// TIA Portal project "WindTurbineOperativeState" (V17)
// Operation state control system of wind turbine

(* hardware
DEVICE "S7-1200 station_1"  S7-1200 Station
   slot 0: "Rack_0"  S7-1200 Rack  Rack  V1.0
   slot 1: "PLC_1"  CPU 1211C DC/DC/DC  6ES7 211-1AE40-0XB0  V4.5
*)

// ===== PLC "PLC_1"  CPU 1211C DC/DC/DC =====

VAR_GLOBAL   // PLC tag table "Default tag table"
   "_WindSpeed_AI" AT %IW64 : Int;
   "_TurbineRotation_AI" AT %IW66 : Int;
   "EmergencyStop_BTN" AT %I0.0 : Bool;
   "BlockState_BTN" AT %I0.1 : Bool;
   "ParkingBrake" AT %Q0.0 : Bool;
   "PitchBrake" AT %Q0.1 : Bool;
   "GeneratorTrip" AT %Q0.2 : Bool;
   "_BlockState" AT %M0.0 : Bool;
   "WebError" AT %MW0 : Int;
END_VAR

VAR_GLOBAL CONSTANT   // PLC tag table "Default tag table"
   "_ParkBrake" : Byte := 0;
   "_Startup" : Byte := 1;
   "_Generating" : Byte := 2;
   "_PitchBrake" : Byte := 3;
END_VAR

DATA_BLOCK "CompOnDuration_DB_13"   // DB1
{ S7_Optimized_Access := 'TRUE' }
VERSION : 0.1
// stored: InstanceOfName CompOnDuration
"CompOnDuration"
BEGIN
END_DATA_BLOCK

DATA_BLOCK "CompOnDuration_DB_01"   // DB2
{ S7_Optimized_Access := 'TRUE' }
VERSION : 0.1
// stored: InstanceOfName CompOnDuration
"CompOnDuration"
BEGIN
END_DATA_BLOCK

DATA_BLOCK "CompOnDuration_DB_02"   // DB3
{ S7_Optimized_Access := 'TRUE' }
VERSION : 0.1
// stored: InstanceOfName CompOnDuration
"CompOnDuration"
BEGIN
END_DATA_BLOCK

DATA_BLOCK "CompOnDuration_DB_03"   // DB4
{ S7_Optimized_Access := 'TRUE' }
VERSION : 0.1
// stored: InstanceOfName CompOnDuration
"CompOnDuration"
BEGIN
END_DATA_BLOCK

DATA_BLOCK "CompOnDuration_DB_04"   // DB5
{ S7_Optimized_Access := 'TRUE' }
VERSION : 0.1
// stored: InstanceOfName CompOnDuration
"CompOnDuration"
BEGIN
END_DATA_BLOCK

DATA_BLOCK "CompOnDuration_DB_05"   // DB6
{ S7_Optimized_Access := 'TRUE' }
VERSION : 0.1
// stored: InstanceOfName CompOnDuration
"CompOnDuration"
BEGIN
END_DATA_BLOCK

DATA_BLOCK "CompOnDuration_DB_06"   // DB7
{ S7_Optimized_Access := 'TRUE' }
VERSION : 0.1
// stored: InstanceOfName CompOnDuration
"CompOnDuration"
BEGIN
END_DATA_BLOCK

DATA_BLOCK "CompOnDuration_DB_07"   // DB8
{ S7_Optimized_Access := 'TRUE' }
VERSION : 0.1
// stored: InstanceOfName CompOnDuration
"CompOnDuration"
BEGIN
END_DATA_BLOCK

DATA_BLOCK "CompOnDuration_DB_08"   // DB9
{ S7_Optimized_Access := 'TRUE' }
VERSION : 0.1
// stored: InstanceOfName CompOnDuration
"CompOnDuration"
BEGIN
END_DATA_BLOCK

DATA_BLOCK "CompOnDuration_DB_09"   // DB10
{ S7_Optimized_Access := 'TRUE' }
VERSION : 0.1
// stored: InstanceOfName CompOnDuration
"CompOnDuration"
BEGIN
END_DATA_BLOCK

DATA_BLOCK "CompOnDuration_DB_10"   // DB11
{ S7_Optimized_Access := 'TRUE' }
VERSION : 0.1
// stored: InstanceOfName CompOnDuration
"CompOnDuration"
BEGIN
END_DATA_BLOCK

DATA_BLOCK "CompOnDuration_DB_11"   // DB12
{ S7_Optimized_Access := 'TRUE' }
VERSION : 0.1
// stored: InstanceOfName CompOnDuration
"CompOnDuration"
BEGIN
END_DATA_BLOCK

DATA_BLOCK "CompOnDuration_DB_12"   // DB13
{ S7_Optimized_Access := 'TRUE' }
VERSION : 0.1
// stored: InstanceOfName CompOnDuration
"CompOnDuration"
BEGIN
END_DATA_BLOCK

DATA_BLOCK "ModBus_DB"   // DB14
{ S7_Optimized_Access := 'TRUE' }
VERSION : 0.1
   VAR
      CONNECT : TCON_IP_v4;
      ERROR : Bool;
      STATUS : Word;
   END_VAR
BEGIN
   CONNECT.InterfaceId := 64;
   CONNECT.LocalPort := 502;
   CONNECT.ID := 1;
   CONNECT.ConnectionType := 11;
END_DATA_BLOCK

DATA_BLOCK "Hold_Reg"   // DB16
{ S7_Optimized_Access := 'FALSE' }
VERSION : 0.1
   VAR
      TurbineState : Byte;
      BlockState_MB : Bool := false;
      vWind : Real;
      wTurbine : Real;
      vWind_CutInLow : Real := 4.0;
      vWind_CutInUp : Real := 18.0;
      vWind_CutOut : Real := 20.0;
      wTurbine_CutIn : Real := 11.0;
      wTurbine_CutOut : Real := 22.0;
      wTurbine_Parking : Real := 2.0;
      vWind_zero : Int := 34;   // Ofset for 0 reference dac0
      vWind_max : Int := 25051;   // Ofset for 1023 reference dac0
      vWind_gain : Real := 102.3;   // Scale to SI value for "vWind_AI"
      wTurbine_zero : Int := 0;   // Ofset for 0 reference dac1
      wTurbine_max : Int := 25151;   // Ofset for 1023 reference dac1
      wTurbine_gain : Real := 31.0;   // Scale to SI value for "wTurbine_AI"
      time_0 : Time := T#700ms;
      time_1 : Time := T#1.5s;
      time_2 : Time := T#3s;
   END_VAR
BEGIN
END_DATA_BLOCK

FUNCTION_BLOCK "CompOnDuration"   // FB1, LAD
{ S7_Optimized_Access := 'TRUE' }
VERSION : 0.1
// Compare if #A > #B for a duration of at least #Time set #Q
   VAR_INPUT
      "A" : Real;
      "B" : Real;
      "Time" : Time;
   END_VAR
   VAR_OUTPUT
      Q : Bool;
   END_VAR
   VAR
      "IEC_Timer_Multi-Instance" : TON_TIME;
   END_VAR
BEGIN

REGION Network 1
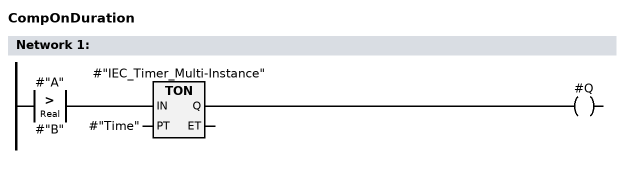
   #"IEC_Timer_Multi-Instance"(IN := #"A" > #"B", PT := #"Time");   // TON
   #Q := #"IEC_Timer_Multi-Instance".Q;
END_REGION
END_FUNCTION_BLOCK

ORGANIZATION_BLOCK "Main"   // OB1, LAD, ProgramCycle
TITLE = "Main Program Sweep (Cycle)"
{ S7_Optimized_Access := 'TRUE' }
VERSION : 0.1
// State machine turbine operation
   VAR_INPUT
      Initial_Call : Bool;   // Initial call of this OB
      Remanence : Bool;   // =True, if remanent data are available
   END_VAR
   VAR_TEMP
      "0to1_1" : Bool;
      "0to1_2" : Bool;
      "1to2" : Bool;
      "1to3_1" : Bool;
      "1to3_2" : Bool;
      "2to3_1" : Bool;
      "2to3_2" : Bool;
      "2to3_3" : Bool;
      "2to3_4" : Bool;
      "3to1_1" : Bool;
      "3to1_2" : Bool;
      "3to1_3" : Bool;
      "3to0" : Bool;
      Norm_vWind : Real;
      Norm_wTurbine : Real;
   END_VAR
   VAR_TEMP   // added for the SCL form of the ladder/FBD networks
      _w1 : Bool;
      _w2 : Bool;
      _w3 : Bool;
      _w4 : Bool;
   END_VAR
BEGIN

REGION Network 1: vWind conversion
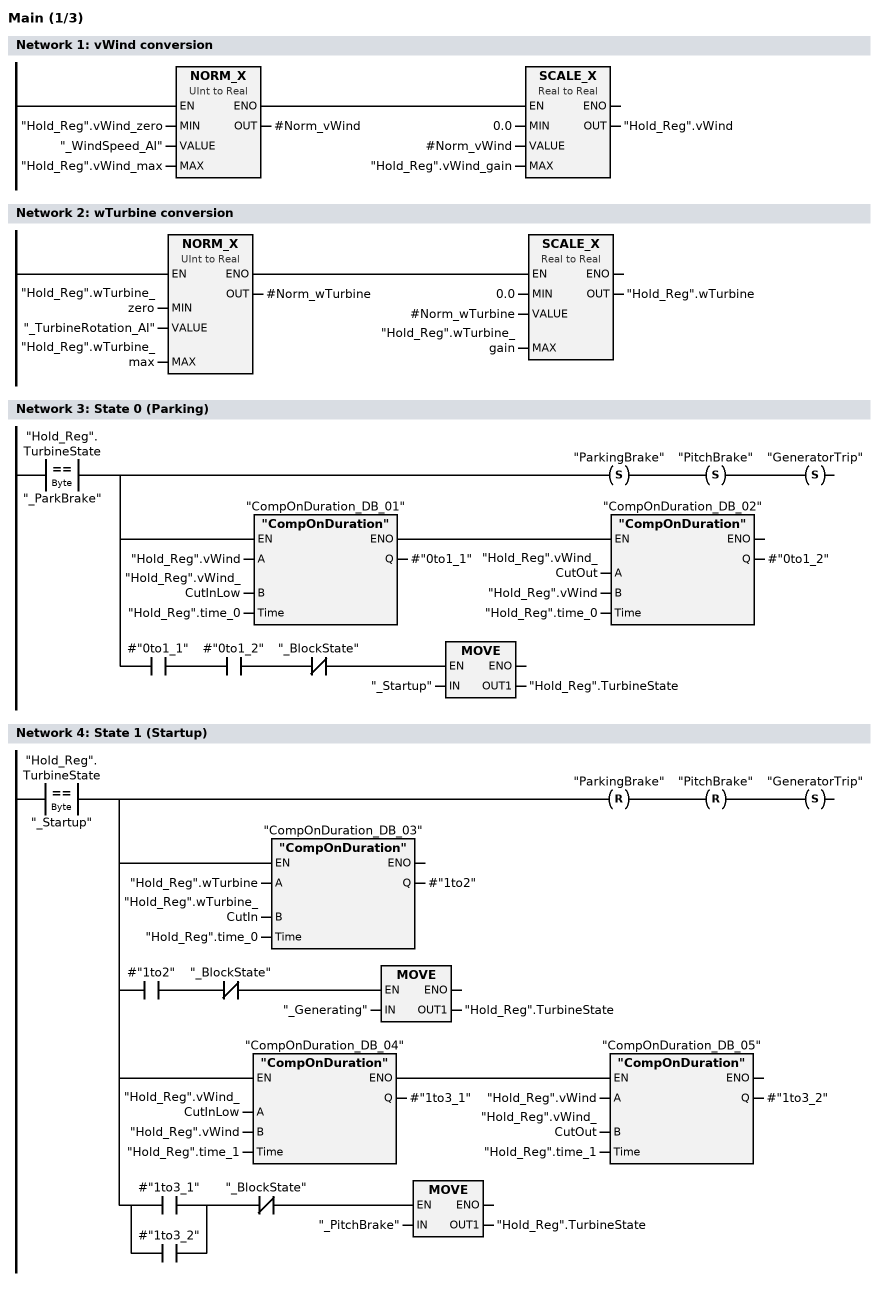
   RUNG wire#powerrail
      { S7_Templates := "[SrcType := UInt, DestType := Real]" } Normalize(min := "Hold_Reg".vWind_zero, value := "_WindSpeed_AI", max := "Hold_Reg".vWind_max, out => #Norm_vWind)
      { S7_Templates := "[SrcType := Real, DestType := Real]" } Scale(min := 0.0, value := #Norm_vWind, max := "Hold_Reg".vWind_gain, out => "Hold_Reg".vWind)
   END_RUNG
   // the same network as SCL:
   #Norm_vWind := NORM_X(MIN := "Hold_Reg".vWind_zero, VALUE := "_WindSpeed_AI", MAX := "Hold_Reg".vWind_max);
   "Hold_Reg".vWind := SCALE_X(MIN := 0.0, VALUE := #Norm_vWind, MAX := "Hold_Reg".vWind_gain);
END_REGION

REGION Network 2: wTurbine conversion
   RUNG wire#powerrail
      { S7_Templates := "[SrcType := UInt, DestType := Real]" } Normalize(min := "Hold_Reg".wTurbine_zero, value := "_TurbineRotation_AI", max := "Hold_Reg".wTurbine_max, out => #Norm_wTurbine)
      { S7_Templates := "[SrcType := Real, DestType := Real]" } Scale(min := 0.0, value := #Norm_wTurbine, max := "Hold_Reg".wTurbine_gain, out => "Hold_Reg".wTurbine)
   END_RUNG
   // the same network as SCL:
   #Norm_wTurbine := NORM_X(MIN := "Hold_Reg".wTurbine_zero, VALUE := "_TurbineRotation_AI", MAX := "Hold_Reg".wTurbine_max);
   "Hold_Reg".wTurbine := SCALE_X(MIN := 0.0, VALUE := #Norm_wTurbine, MAX := "Hold_Reg".wTurbine_gain);
END_REGION

REGION Network 3: State 0 (Parking)
   RUNG wire#powerrail
      { S7_Templates := "SrcType := Byte" } EQ_Contact(in1 := "Hold_Reg".TurbineState, in2 := "_ParkBrake")
      wire#w1
      S_Coil( "ParkingBrake" )
      S_Coil( "PitchBrake" )
      S_Coil( "GeneratorTrip" )
   END_RUNG
   RUNG wire#w1
      "CompOnDuration_DB_01"("A" := "Hold_Reg".vWind, "B" := "Hold_Reg".vWind_CutInLow, "Time" := "Hold_Reg".time_0, Q => #"0to1_1")
      "CompOnDuration_DB_02"("A" := "Hold_Reg".vWind_CutOut, "B" := "Hold_Reg".vWind, "Time" := "Hold_Reg".time_0, Q => #"0to1_2")
   END_RUNG
   RUNG wire#w1
      Contact( #"0to1_1" )
      Contact( #"0to1_2" )
      I_Contact( "_BlockState" )
      Move(in := "_Startup", out1 => "Hold_Reg".TurbineState)
   END_RUNG
   // the same network as SCL:
   #_w1 := "Hold_Reg".TurbineState = "_ParkBrake";
   IF #_w1 THEN
       "ParkingBrake" := TRUE;
       "PitchBrake" := TRUE;
       "GeneratorTrip" := TRUE;
   END_IF;
   "CompOnDuration_DB_01"(EN := #_w1,   // "CompOnDuration"
                          "A" := "Hold_Reg".vWind,
                          "B" := "Hold_Reg".vWind_CutInLow,
                          "Time" := "Hold_Reg".time_0,
                          Q => #"0to1_1",
                          ENO => #_w2);
   IF #_w2 THEN
       "CompOnDuration_DB_02"("A" := "Hold_Reg".vWind_CutOut,   // "CompOnDuration"
                              "B" := "Hold_Reg".vWind,
                              "Time" := "Hold_Reg".time_0,
                              Q => #"0to1_2");
   END_IF;
   IF #_w1 AND #"0to1_1" AND #"0to1_2" AND NOT "_BlockState" THEN
       "Hold_Reg".TurbineState := "_Startup";
   END_IF;
END_REGION

REGION Network 4: State 1 (Startup)
   RUNG wire#powerrail
      { S7_Templates := "SrcType := Byte" } EQ_Contact(in1 := "Hold_Reg".TurbineState, in2 := "_Startup")
      wire#w1
      R_Coil( "ParkingBrake" )
      R_Coil( "PitchBrake" )
      S_Coil( "GeneratorTrip" )
   END_RUNG
   RUNG wire#w1
      "CompOnDuration_DB_03"("A" := "Hold_Reg".wTurbine, "B" := "Hold_Reg".wTurbine_CutIn, "Time" := "Hold_Reg".time_0, Q => #"1to2")
   END_RUNG
   RUNG wire#w1
      Contact( #"1to2" )
      I_Contact( "_BlockState" )
      Move(in := "_Generating", out1 => "Hold_Reg".TurbineState)
   END_RUNG
   RUNG wire#w1
      "CompOnDuration_DB_04"("A" := "Hold_Reg".vWind_CutInLow, "B" := "Hold_Reg".vWind, "Time" := "Hold_Reg".time_1, Q => #"1to3_1")
      "CompOnDuration_DB_05"("A" := "Hold_Reg".vWind, "B" := "Hold_Reg".vWind_CutOut, "Time" := "Hold_Reg".time_1, Q => #"1to3_2")
   END_RUNG
   RUNG wire#w1
      Contact( #"1to3_1" )
      wire#w2
      I_Contact( "_BlockState" )
      Move(in := "_PitchBrake", out1 => "Hold_Reg".TurbineState)
   END_RUNG
   RUNG wire#w1
      Contact( #"1to3_2" )
   END_RUNG wire#w2
   // the same network as SCL:
   #_w1 := "Hold_Reg".TurbineState = "_Startup";
   IF #_w1 THEN
       "ParkingBrake" := FALSE;
       "PitchBrake" := FALSE;
       "GeneratorTrip" := TRUE;
       "CompOnDuration_DB_03"("A" := "Hold_Reg".wTurbine,   // "CompOnDuration"
                              "B" := "Hold_Reg".wTurbine_CutIn,
                              "Time" := "Hold_Reg".time_0,
                              Q => #"1to2");
   END_IF;
   IF #_w1 AND #"1to2" AND NOT "_BlockState" THEN "Hold_Reg".TurbineState := "_Generating"; END_IF;
   "CompOnDuration_DB_04"(EN := #_w1,   // "CompOnDuration"
                          "A" := "Hold_Reg".vWind_CutInLow,
                          "B" := "Hold_Reg".vWind,
                          "Time" := "Hold_Reg".time_1,
                          Q => #"1to3_1",
                          ENO => #_w2);
   IF #_w2 THEN
       "CompOnDuration_DB_05"("A" := "Hold_Reg".vWind,   // "CompOnDuration"
                              "B" := "Hold_Reg".vWind_CutOut,
                              "Time" := "Hold_Reg".time_1,
                              Q => #"1to3_2");
   END_IF;
   IF #_w1 AND (#"1to3_1" OR #"1to3_2") AND NOT "_BlockState" THEN
       "Hold_Reg".TurbineState := "_PitchBrake";
   END_IF;
END_REGION

REGION Network 5: State 2 (Generating)
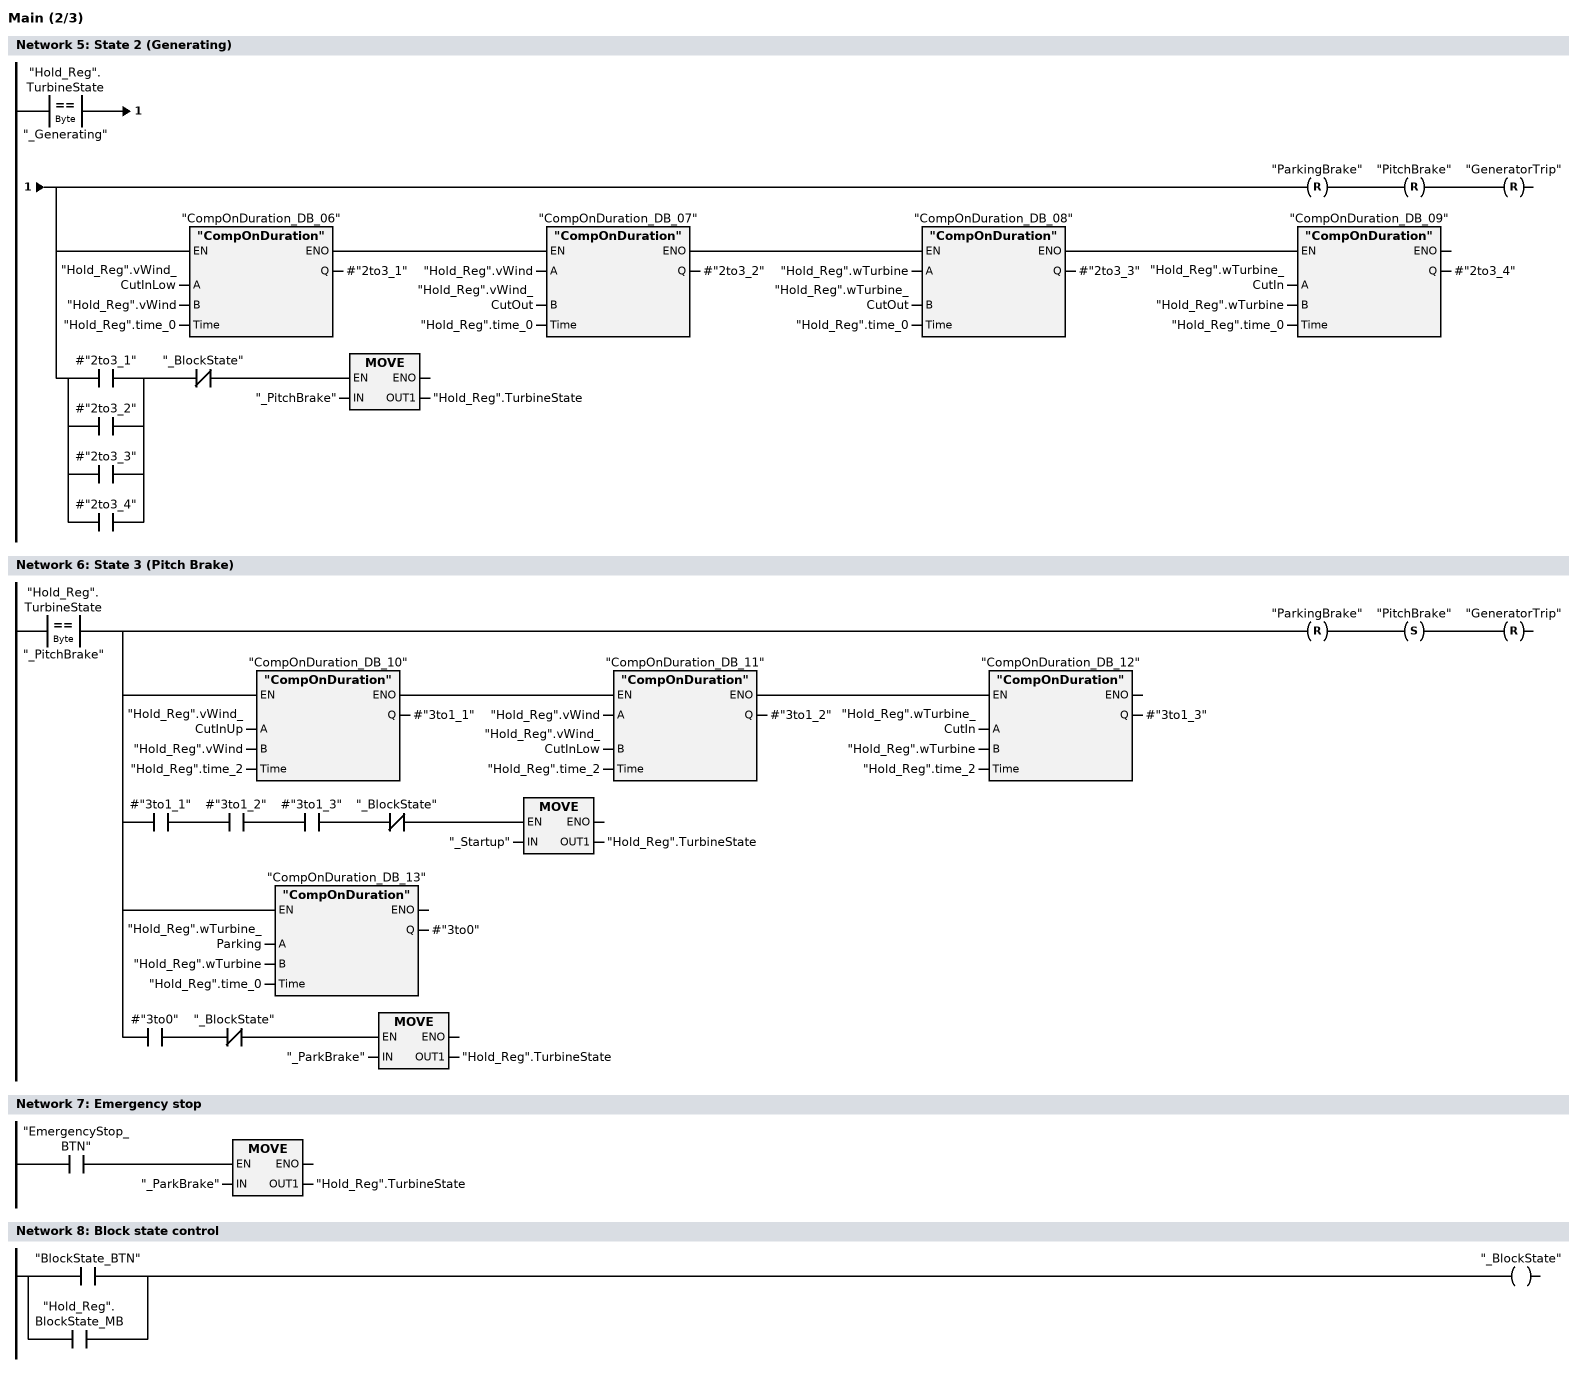
   RUNG wire#powerrail
      { S7_Templates := "SrcType := Byte" } EQ_Contact(in1 := "Hold_Reg".TurbineState, in2 := "_Generating")
      wire#w1
      R_Coil( "ParkingBrake" )
      R_Coil( "PitchBrake" )
      R_Coil( "GeneratorTrip" )
   END_RUNG
   RUNG wire#w1
      "CompOnDuration_DB_06"("A" := "Hold_Reg".vWind_CutInLow, "B" := "Hold_Reg".vWind, "Time" := "Hold_Reg".time_0, Q => #"2to3_1")
      "CompOnDuration_DB_07"("A" := "Hold_Reg".vWind, "B" := "Hold_Reg".vWind_CutOut, "Time" := "Hold_Reg".time_0, Q => #"2to3_2")
      "CompOnDuration_DB_08"("A" := "Hold_Reg".wTurbine, "B" := "Hold_Reg".wTurbine_CutOut, "Time" := "Hold_Reg".time_0, Q => #"2to3_3")
      "CompOnDuration_DB_09"("A" := "Hold_Reg".wTurbine_CutIn, "B" := "Hold_Reg".wTurbine, "Time" := "Hold_Reg".time_0, Q => #"2to3_4")
   END_RUNG
   RUNG wire#w1
      Contact( #"2to3_1" )
      wire#w2
      I_Contact( "_BlockState" )
      Move(in := "_PitchBrake", out1 => "Hold_Reg".TurbineState)
   END_RUNG
   RUNG wire#w1
      Contact( #"2to3_2" )
   END_RUNG wire#w2
   RUNG wire#w1
      Contact( #"2to3_3" )
   END_RUNG wire#w2
   RUNG wire#w1
      Contact( #"2to3_4" )
   END_RUNG wire#w2
   // the same network as SCL:
   #_w1 := "Hold_Reg".TurbineState = "_Generating";
   IF #_w1 THEN
       "ParkingBrake" := FALSE;
       "PitchBrake" := FALSE;
       "GeneratorTrip" := FALSE;
   END_IF;
   "CompOnDuration_DB_06"(EN := #_w1,   // "CompOnDuration"
                          "A" := "Hold_Reg".vWind_CutInLow,
                          "B" := "Hold_Reg".vWind,
                          "Time" := "Hold_Reg".time_0,
                          Q => #"2to3_1",
                          ENO => #_w2);
   "CompOnDuration_DB_07"(EN := #_w2,   // "CompOnDuration"
                          "A" := "Hold_Reg".vWind,
                          "B" := "Hold_Reg".vWind_CutOut,
                          "Time" := "Hold_Reg".time_0,
                          Q => #"2to3_2",
                          ENO => #_w3);
   "CompOnDuration_DB_08"(EN := #_w3,   // "CompOnDuration"
                          "A" := "Hold_Reg".wTurbine,
                          "B" := "Hold_Reg".wTurbine_CutOut,
                          "Time" := "Hold_Reg".time_0,
                          Q => #"2to3_3",
                          ENO => #_w4);
   IF #_w4 THEN
       "CompOnDuration_DB_09"("A" := "Hold_Reg".wTurbine_CutIn,   // "CompOnDuration"
                              "B" := "Hold_Reg".wTurbine,
                              "Time" := "Hold_Reg".time_0,
                              Q => #"2to3_4");
   END_IF;
   IF #_w1 AND (#"2to3_1" OR #"2to3_2" OR #"2to3_3" OR #"2to3_4") AND NOT "_BlockState" THEN
       "Hold_Reg".TurbineState := "_PitchBrake";
   END_IF;
END_REGION

REGION Network 6: State 3 (Pitch Brake)
   RUNG wire#powerrail
      { S7_Templates := "SrcType := Byte" } EQ_Contact(in1 := "Hold_Reg".TurbineState, in2 := "_PitchBrake")
      wire#w1
      R_Coil( "ParkingBrake" )
      S_Coil( "PitchBrake" )
      R_Coil( "GeneratorTrip" )
   END_RUNG
   RUNG wire#w1
      "CompOnDuration_DB_10"("A" := "Hold_Reg".vWind_CutInUp, "B" := "Hold_Reg".vWind, "Time" := "Hold_Reg".time_2, Q => #"3to1_1")
      "CompOnDuration_DB_11"("A" := "Hold_Reg".vWind, "B" := "Hold_Reg".vWind_CutInLow, "Time" := "Hold_Reg".time_2, Q => #"3to1_2")
      "CompOnDuration_DB_12"("A" := "Hold_Reg".wTurbine_CutIn, "B" := "Hold_Reg".wTurbine, "Time" := "Hold_Reg".time_2, Q => #"3to1_3")
   END_RUNG
   RUNG wire#w1
      Contact( #"3to1_1" )
      Contact( #"3to1_2" )
      Contact( #"3to1_3" )
      I_Contact( "_BlockState" )
      Move(in := "_Startup", out1 => "Hold_Reg".TurbineState)
   END_RUNG
   RUNG wire#w1
      "CompOnDuration_DB_13"("A" := "Hold_Reg".wTurbine_Parking, "B" := "Hold_Reg".wTurbine, "Time" := "Hold_Reg".time_0, Q => #"3to0")
   END_RUNG
   RUNG wire#w1
      Contact( #"3to0" )
      I_Contact( "_BlockState" )
      Move(in := "_ParkBrake", out1 => "Hold_Reg".TurbineState)
   END_RUNG
   // the same network as SCL:
   #_w1 := "Hold_Reg".TurbineState = "_PitchBrake";
   IF #_w1 THEN
       "ParkingBrake" := FALSE;
       "PitchBrake" := TRUE;
       "GeneratorTrip" := FALSE;
   END_IF;
   "CompOnDuration_DB_10"(EN := #_w1,   // "CompOnDuration"
                          "A" := "Hold_Reg".vWind_CutInUp,
                          "B" := "Hold_Reg".vWind,
                          "Time" := "Hold_Reg".time_2,
                          Q => #"3to1_1",
                          ENO => #_w2);
   "CompOnDuration_DB_11"(EN := #_w2,   // "CompOnDuration"
                          "A" := "Hold_Reg".vWind,
                          "B" := "Hold_Reg".vWind_CutInLow,
                          "Time" := "Hold_Reg".time_2,
                          Q => #"3to1_2",
                          ENO => #_w3);
   IF #_w3 THEN
       "CompOnDuration_DB_12"("A" := "Hold_Reg".wTurbine_CutIn,   // "CompOnDuration"
                              "B" := "Hold_Reg".wTurbine,
                              "Time" := "Hold_Reg".time_2,
                              Q => #"3to1_3");
   END_IF;
   IF #_w1 AND #"3to1_1" AND #"3to1_2" AND #"3to1_3" AND NOT "_BlockState" THEN
       "Hold_Reg".TurbineState := "_Startup";
   END_IF;
   IF #_w1 THEN
       "CompOnDuration_DB_13"("A" := "Hold_Reg".wTurbine_Parking,   // "CompOnDuration"
                              "B" := "Hold_Reg".wTurbine,
                              "Time" := "Hold_Reg".time_0,
                              Q => #"3to0");
   END_IF;
   IF #_w1 AND #"3to0" AND NOT "_BlockState" THEN "Hold_Reg".TurbineState := "_ParkBrake"; END_IF;
END_REGION

REGION Network 7: Emergency stop
   RUNG wire#powerrail
      Contact( "EmergencyStop_BTN" )
      Move(in := "_ParkBrake", out1 => "Hold_Reg".TurbineState)
   END_RUNG
   // the same network as SCL:
   IF "EmergencyStop_BTN" THEN "Hold_Reg".TurbineState := "_ParkBrake"; END_IF;
END_REGION

REGION Network 8: Block state control
   RUNG wire#powerrail
      Contact( "BlockState_BTN" )
      wire#w1
      Coil( "_BlockState" )
   END_RUNG
   RUNG wire#powerrail
      Contact( "Hold_Reg".BlockState_MB )
   END_RUNG wire#w1
   // the same network as SCL:
   "_BlockState" := "BlockState_BTN" OR "Hold_Reg".BlockState_MB;
END_REGION

REGION Network 9: Modbus server
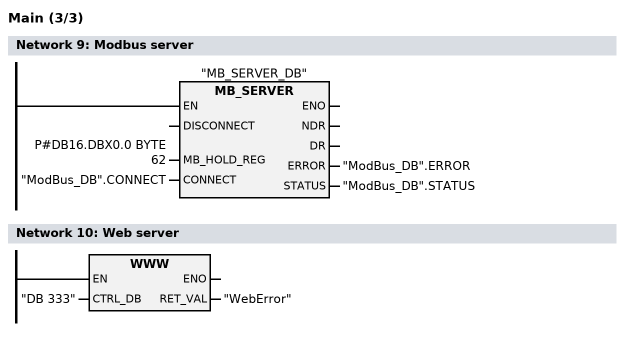
   "MB_SERVER_DB"(MB_HOLD_REG := P#DB16.DBX0.0 BYTE 62,   // MB_SERVER
                  CONNECT := "ModBus_DB".CONNECT,
                  ERROR => "ModBus_DB".ERROR,
                  STATUS => "ModBus_DB".STATUS);
END_REGION

REGION Network 10: Web server
   "WebError" := WWW(CTRL_DB := "DB 333");
END_REGION
END_ORGANIZATION_BLOCK